KUKA KRL data list: AbreGarra.dat

&ACCESS RVO1
&REL 1
&PARAM EDITMASK = *
DEFDAT AbreGarra

ENDDAT
